FUNCTION_BLOCK ML_model
  (* Version 1.0, 2005-07-27, Goran Cengic, Chalmers *)
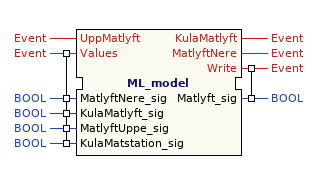
  EVENT_INPUT
    UppMatlyft;
    Values WITH MatlyftNere_sig, KulaMatlyft_sig, MatlyftUppe_sig, KulaMatstation_sig;
  END_EVENT
  EVENT_OUTPUT
    KulaMatlyft;
    MatlyftNere;
    Write WITH Matlyft_sig;
  END_EVENT
  VAR_INPUT
    MatlyftNere_sig : BOOL;
    KulaMatlyft_sig : BOOL;
    MatlyftUppe_sig : BOOL;
    KulaMatstation_sig : BOOL;
  END_VAR
  VAR_OUTPUT
    Matlyft_sig : BOOL;
  END_VAR
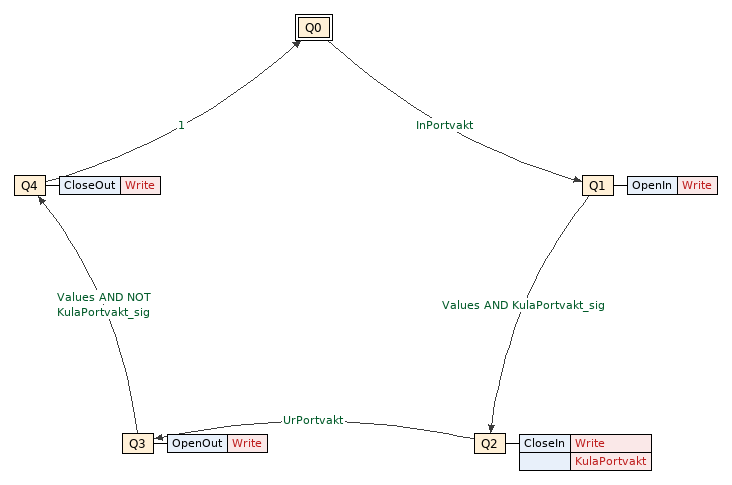
  EC_STATES
    Q0;
    Q1 : OpenIn -> Write;
    Q2 : CloseIn -> Write, -> KulaPortvakt;
    Q3 : OpenOut -> Write;
    Q4 : CloseOut -> Write;
  END_STATES
  EC_TRANSITIONS
    Q0 TO Q1 := InPortvakt;
    Q1 TO Q2 := Values AND KulaPortvakt_sig;
    Q2 TO Q3 := UrPortvakt;
    Q3 TO Q4 := Values AND NOT KulaPortvakt_sig;
    Q4 TO Q0 := 1;
  END_TRANSITIONS
  ALGORITHM OpenIn IN Java:
		System.out.println("Opening Portvakt In.");
		InPortvakt_sig = true;
  END_ALGORITHM
  ALGORITHM CloseIn IN Java:
		System.out.println("Closing Portvakt In.");
		InPortvakt_sig = false;
  END_ALGORITHM
  ALGORITHM OpenOut IN Java:
		System.out.println("Opening Portvakt Out.");
		UrPortvakt_sig = true;
  END_ALGORITHM
  ALGORITHM CloseOut IN Java:
		System.out.println("Closing Portvakt Out.");
		UrPortvakt_sig = false;
  END_ALGORITHM
END_FUNCTION_BLOCK
